// Tests for FB_DigitalOutput. Focus is on the behavior the device exposes
// to callers and HMIs:
//
//   * command routing through F_ValidateRequester (source lock)
//   * request-vs-output bookkeeping (commanded always reflects the
//     latest intent, value always reflects the physical bit)
//   * debounce timers actually gating the output
//   * invert in Regular mode
//   * BAD quality holding the last-known-good output
//   * edge pulses being exactly one scan wide
//   * SinglePulse arming on rising edge and cancelling on commanded LOW
//
// Time-dependent behavior is covered by choosing timer values that either
// clamp to zero (instant fire) or stay effectively infinite for the test
// (T#1S), so a single cyclic call lands in the branch under test without
// waiting real time.
FUNCTION_BLOCK FB_DigitalOutput_Test EXTENDS TcUnit.FB_TestSuite

InitialStateReady();
SetOnFromProgDrivesOutputHigh();
SetOffAfterSetOnDrivesOutputLow();
SetOnAcceptedFromProgEvenWhenLocked();
SetOnRejectedFromOperatorWhenLocked();
DebounceOnBlocksOutputUntilElapsed();
DebounceOffHoldsOutputHighUntilElapsed();
InvertFlipsOutputInRegularMode();
BadQualityHoldsLastKnownGoodOutput();
StsCommandedMirrorsRequestEvenUnderBadQuality();
EdgePulsesAreOneScanWide();
SinglePulseFiresOnCommandAndCanBeCanceled();

METHOD InitialStateReady
VAR
    fb : TcForge.FB_DigitalOutput;
END_VAR
TEST('InitialStateReady');

// Fresh instance + one good-quality cycle: no commands issued, no faults
// raised, output dead.
fb(inpQuality := TcForge.E_IO_Quality.GOOD);

AssertFalse(
    Condition := fb.sts.value,
    Message   := 'Fresh instance must start with physical output LOW');
AssertFalse(
    Condition := fb.sts.commanded,
    Message   := 'Fresh instance must start with commanded request LOW');
AssertFalse(
    Condition := fb.sts.header.faulted,
    Message   := 'Fresh instance must not be faulted');
AssertTrue(
    Condition := fb.sts.header.ready,
    Message   := 'Fresh instance must report ready TRUE (no fault, not busy, not locked)');
AssertFalse(
    Condition := fb.sts.header.sourceLocked,
    Message   := 'Fresh instance must not be source-locked');

TEST_FINISHED();
END_METHOD

METHOD SetOnFromProgDrivesOutputHigh
VAR
    fb     : TcForge.FB_DigitalOutput;
    resp   : TcForge.E_RpcMethodResponse;
END_VAR
TEST('SetOnFromProgDrivesOutputHigh');

// Default cfg: no debounce (PT = T#0MS), Regular mode, no invert.
// A single SetOn + one cycle should flush straight through to the
// physical output.
resp := fb.SetOn(eRequester := TcForge.E_Requester.PROG);
fb(inpQuality := TcForge.E_IO_Quality.GOOD);

AssertEquals_DINT(
    Expected := TcForge.E_RpcMethodResponse.ACCEPTED,
    Actual   := resp,
    Message  := 'SetOn from PROG on a fresh instance must be ACCEPTED');
AssertTrue(
    Condition := fb.sts.value,
    Message   := 'Regular mode with no debounce must flush SetOn to the physical output in one cycle');
AssertTrue(
    Condition := fb.sts.commanded,
    Message   := 'commanded must reflect the accepted SetOn request');

TEST_FINISHED();
END_METHOD

METHOD SetOffAfterSetOnDrivesOutputLow
VAR
    fb   : TcForge.FB_DigitalOutput;
    resp : TcForge.E_RpcMethodResponse;
END_VAR
TEST('SetOffAfterSetOnDrivesOutputLow');

fb.SetOn(eRequester := TcForge.E_Requester.PROG);
fb(inpQuality := TcForge.E_IO_Quality.GOOD);

resp := fb.SetOff(eRequester := TcForge.E_Requester.PROG);
fb(inpQuality := TcForge.E_IO_Quality.GOOD);

AssertEquals_DINT(
    Expected := TcForge.E_RpcMethodResponse.ACCEPTED,
    Actual   := resp,
    Message  := 'SetOff from PROG must be ACCEPTED');
AssertFalse(
    Condition := fb.sts.value,
    Message   := 'SetOff must drop the physical output LOW in one cycle with no debounce');
AssertFalse(
    Condition := fb.sts.commanded,
    Message   := 'commanded must follow the latest SetOff request');

TEST_FINISHED();
END_METHOD

METHOD SetOnAcceptedFromProgEvenWhenLocked
VAR
    fb   : TcForge.FB_DigitalOutput;
    resp : TcForge.E_RpcMethodResponse;
END_VAR
TEST('SetOnAcceptedFromProgEvenWhenLocked');

// bSourceLockedToProg is meant to gate OPERATOR; PROG must always get
// through so the program can still drive the output after locking out the
// operator.
fb.LockSource(bLock := TRUE);
resp := fb.SetOn(eRequester := TcForge.E_Requester.PROG);
fb(inpQuality := TcForge.E_IO_Quality.GOOD);

AssertEquals_DINT(
    Expected := TcForge.E_RpcMethodResponse.ACCEPTED,
    Actual   := resp,
    Message  := 'PROG requester must be accepted even with source-lock active');
AssertTrue(
    Condition := fb.sts.value,
    Message   := 'Accepted SetOn from PROG must still drive the physical output');
AssertTrue(
    Condition := fb.sts.header.sourceLocked,
    Message   := 'header must reflect source-lock state');

TEST_FINISHED();
END_METHOD

METHOD SetOnRejectedFromOperatorWhenLocked
VAR
    fb   : TcForge.FB_DigitalOutput;
    resp : TcForge.E_RpcMethodResponse;
END_VAR
TEST('SetOnRejectedFromOperatorWhenLocked');

fb.LockSource(bLock := TRUE);
resp := fb.SetOn(eRequester := TcForge.E_Requester.OPERATOR);
fb(inpQuality := TcForge.E_IO_Quality.GOOD);

AssertEquals_DINT(
    Expected := TcForge.E_RpcMethodResponse.REJECTED_SOURCE_NOT_ALLOWED,
    Actual   := resp,
    Message  := 'OPERATOR requester must be rejected while source-locked');
AssertFalse(
    Condition := fb.sts.value,
    Message   := 'Rejected SetOn must not touch the physical output');
AssertFalse(
    Condition := fb.sts.commanded,
    Message   := 'Rejected SetOn must not update commanded');

TEST_FINISHED();
END_METHOD

METHOD DebounceOnBlocksOutputUntilElapsed
VAR
    fb : TcForge.FB_DigitalOutput;
END_VAR
TEST('DebounceOnBlocksOutputUntilElapsed');

// debounceOn = T#1S — far longer than this synchronous test will run,
// so _tonOn.Q must still be FALSE when we check: the output must be held
// LOW while the debounce hasn't elapsed.
fb.cfg.debounceOn := T#1S;
fb.SetOn(eRequester := TcForge.E_Requester.PROG);
fb(inpQuality := TcForge.E_IO_Quality.GOOD);

AssertTrue(
    Condition := fb.sts.commanded,
    Message   := 'commanded must reflect the request immediately (debounce gates the output, not the request)');
AssertFalse(
    Condition := fb.sts.value,
    Message   := 'debounceOn must hold the physical output LOW until the TON elapses');

TEST_FINISHED();
END_METHOD

METHOD DebounceOffHoldsOutputHighUntilElapsed
VAR
    fb : TcForge.FB_DigitalOutput;
END_VAR
TEST('DebounceOffHoldsOutputHighUntilElapsed');

// debounceOn stays at 0 so the output flushes HIGH immediately. The
// OFF-debounce (T#1S) then holds it HIGH even after SetOff, until TOF.Q
// falls — which it will not inside this synchronous test.
fb.cfg.debounceOff := T#1S;
fb.SetOn(eRequester := TcForge.E_Requester.PROG);
fb(inpQuality := TcForge.E_IO_Quality.GOOD);

AssertTrue(
    Condition := fb.sts.value,
    Message   := 'Precondition: SetOn with zero ON-debounce must flush HIGH');

fb.SetOff(eRequester := TcForge.E_Requester.PROG);
fb(inpQuality := TcForge.E_IO_Quality.GOOD);

AssertFalse(
    Condition := fb.sts.commanded,
    Message   := 'commanded must follow the SetOff request regardless of debounce');
AssertTrue(
    Condition := fb.sts.value,
    Message   := 'debounceOff must hold the physical output HIGH until the TOF expires');

TEST_FINISHED();
END_METHOD

METHOD InvertFlipsOutputInRegularMode
VAR
    fb : TcForge.FB_DigitalOutput;
END_VAR
TEST('InvertFlipsOutputInRegularMode');

// Active-low actuator: invert means "commanded ON -> physical LOW".
fb.cfg.invert := TRUE;
fb.SetOn(eRequester := TcForge.E_Requester.PROG);
fb(inpQuality := TcForge.E_IO_Quality.GOOD);

AssertTrue(
    Condition := fb.sts.commanded,
    Message   := 'commanded must reflect logical intent, not inverted physical output');
AssertFalse(
    Condition := fb.sts.value,
    Message   := 'invert must flip HIGH intent into a LOW physical output');

fb.SetOff(eRequester := TcForge.E_Requester.PROG);
fb(inpQuality := TcForge.E_IO_Quality.GOOD);

AssertFalse(
    Condition := fb.sts.commanded,
    Message   := 'commanded must follow SetOff regardless of invert');
AssertTrue(
    Condition := fb.sts.value,
    Message   := 'invert must flip LOW intent into a HIGH physical output');

TEST_FINISHED();
END_METHOD

METHOD BadQualityHoldsLastKnownGoodOutput
VAR
    fb : TcForge.FB_DigitalOutput;
END_VAR
TEST('BadQualityHoldsLastKnownGoodOutput');
fb.cfg.holdOnBadQuality := TRUE;

// Establish HIGH under GOOD quality.
fb.SetOn(eRequester := TcForge.E_Requester.PROG);
fb(inpQuality := TcForge.E_IO_Quality.GOOD);
AssertTrue(
    Condition := fb.sts.value,
    Message   := 'Precondition: SetOn under GOOD quality must drive HIGH');

// Now drop to BAD and try to SetOff. The hardware write must be skipped
// so the actuator stays in its last-known-good state.
fb.SetOff(eRequester := TcForge.E_Requester.PROG);
fb(inpQuality := TcForge.E_IO_Quality.BAD);

AssertTrue(
    Condition := fb.sts.value,
    Message   := 'BAD quality must hold the last-known-good physical output (no hardware write)');
AssertEquals_USINT(
    Expected := TcForge.E_IO_Quality.BAD,
    Actual   := fb.sts.quality,
    Message  := 'quality must surface the BAD tag to downstream consumers');

TEST_FINISHED();
END_METHOD

METHOD StsCommandedMirrorsRequestEvenUnderBadQuality
VAR
    fb : TcForge.FB_DigitalOutput;
END_VAR
TEST('StsCommandedMirrorsRequestEvenUnderBadQuality');
fb.cfg.holdOnBadQuality := TRUE;

// Even when the hardware write is vetoed by quality, commanded must
// still echo the live request so HMIs can show "operator asked for OFF
// but the output is held HIGH because quality is BAD".
fb.SetOn(eRequester := TcForge.E_Requester.PROG);
fb(inpQuality := TcForge.E_IO_Quality.GOOD);
fb.SetOff(eRequester := TcForge.E_Requester.PROG);
fb(inpQuality := TcForge.E_IO_Quality.BAD);

AssertFalse(
    Condition := fb.sts.commanded,
    Message   := 'commanded must reflect the current request even when BAD quality blocks the hardware write');
AssertTrue(
    Condition := fb.sts.value,
    Message   := 'value must still show the held physical output');

TEST_FINISHED();
END_METHOD

METHOD EdgePulsesAreOneScanWide
VAR
    fb : TcForge.FB_DigitalOutput;
END_VAR
TEST('EdgePulsesAreOneScanWide');

// Rising-edge pulse appears the cycle the physical output goes HIGH and
// is gone the next cycle.
fb.SetOn(eRequester := TcForge.E_Requester.PROG);
fb(inpQuality := TcForge.E_IO_Quality.GOOD);
AssertTrue(
    Condition := fb.sts.risingEdge,
    Message   := 'risingEdge must fire on the cycle the physical output goes HIGH');
AssertFalse(
    Condition := fb.sts.fallingEdge,
    Message   := 'fallingEdge must stay LOW on a rising edge cycle');

fb(inpQuality := TcForge.E_IO_Quality.GOOD);
AssertFalse(
    Condition := fb.sts.risingEdge,
    Message   := 'risingEdge must be exactly one scan wide');

// Falling edge on the way back down.
fb.SetOff(eRequester := TcForge.E_Requester.PROG);
fb(inpQuality := TcForge.E_IO_Quality.GOOD);
AssertTrue(
    Condition := fb.sts.fallingEdge,
    Message   := 'fallingEdge must fire on the cycle the physical output goes LOW');

fb(inpQuality := TcForge.E_IO_Quality.GOOD);
AssertFalse(
    Condition := fb.sts.fallingEdge,
    Message   := 'fallingEdge must be exactly one scan wide');

TEST_FINISHED();
END_METHOD

METHOD SinglePulseFiresOnCommandAndCanBeCanceled
VAR
    fb : TcForge.FB_DigitalOutput;
END_VAR
TEST('SinglePulseFiresOnCommandAndCanBeCanceled');

// SinglePulse with a long pulse width (T#10S) so the _tonPulseOn.Q
// stays FALSE inside this synchronous test and we observe the pulse
// while it is active.
fb.cfg.mode    := TcForge.E_DigitalOutput_Mode.SinglePulse;
fb.cfg.pulseOn := T#10S;

fb.SetOn(eRequester := TcForge.E_Requester.PROG);
fb(inpQuality := TcForge.E_IO_Quality.GOOD);

AssertTrue(
    Condition := fb.sts.value,
    Message   := 'SinglePulse must arm on the commanded rising edge and drive HIGH while active');

// Commanded LOW must cancel the pulse early — operator safety shortcut.
fb.SetOff(eRequester := TcForge.E_Requester.PROG);
fb(inpQuality := TcForge.E_IO_Quality.GOOD);

AssertFalse(
    Condition := fb.sts.value,
    Message   := 'SetOff must cancel an in-flight SinglePulse immediately');

TEST_FINISHED();
END_METHOD

END_FUNCTION_BLOCK

(* stored: Version 1.1.0.1, ProductVersion 3.1.4026.12
   POU FB_DigitalOutput_Test: Id {b1c2d3e4-f5a6-7890-abcd-000000000800}, SpecialFunc None
   Method InitialStateReady: Id {b1c2d3e4-f5a6-7890-abcd-000000000801}
   Method SetOnFromProgDrivesOutputHigh: Id {b1c2d3e4-f5a6-7890-abcd-000000000802}
   Method SetOffAfterSetOnDrivesOutputLow: Id {b1c2d3e4-f5a6-7890-abcd-000000000803}
   Method SetOnAcceptedFromProgEvenWhenLocked: Id {b1c2d3e4-f5a6-7890-abcd-000000000804}
   Method SetOnRejectedFromOperatorWhenLocked: Id {b1c2d3e4-f5a6-7890-abcd-000000000805}
   Method DebounceOnBlocksOutputUntilElapsed: Id {b1c2d3e4-f5a6-7890-abcd-000000000806}
   Method DebounceOffHoldsOutputHighUntilElapsed: Id {b1c2d3e4-f5a6-7890-abcd-000000000807}
   Method InvertFlipsOutputInRegularMode: Id {b1c2d3e4-f5a6-7890-abcd-000000000808}
   Method BadQualityHoldsLastKnownGoodOutput: Id {b1c2d3e4-f5a6-7890-abcd-000000000809}
   Method StsCommandedMirrorsRequestEvenUnderBadQuality: Id {b1c2d3e4-f5a6-7890-abcd-00000000080a}
   Method EdgePulsesAreOneScanWide: Id {b1c2d3e4-f5a6-7890-abcd-00000000080b}
   Method SinglePulseFiresOnCommandAndCanBeCanceled: Id {b1c2d3e4-f5a6-7890-abcd-00000000080c} *)
